// TIA Portal project "tank_level_control" (V17)

(* hardware
DEVICE "S7-1200 station_1"  S7-1200 Station
   slot 0: "Rack_0"  S7-1200 Rack  Rack  V1.0
   slot 1: "PLC_1"  CPU 1212C AC/DC/Rly  6ES7 212-1BE31-0XB0  V3.0
   slot 2: "DI 16x24VDC/DQ 16xRelay_1"  SM 1223 DI16/DQ16 x relay  6ES7 223-1PL32-0XB0  V2.0
DEVICE "HMI_1"  KTP600 Basic color PN
   slot 0: "HMI_1"  KTP600 Basic color PN  6AV6 647-0AD11-3AX0  12.0.0.0
   slot 1: "HMI_RT_1"  KTP600 Basic color PN  6AV6 647-0AD11-3AX0  12.0.0.0
   slot 5: "HMI_1.IE_CP_1"  PROFINET Interface  12.0.0.0
      slot 1: "PROFINET Interface_1"  PROFINET Interface
         slot 1: "Port_1"  Port
*)

// ===== PLC "PLC_1"  CPU 1212C AC/DC/Rly =====

VAR_GLOBAL   // PLC tag table "Default tag table"
   "OPEN" AT %M0.0 : Bool;
   "CLOSE" AT %M0.1 : Bool;
   "RUNNING" AT %Q0.2 : Bool;   // RUNNING LAMP INDICATOR
   "Tag_1" AT %M1.0 : Bool;
   "LEVEL" AT %MD100 : Real;
   "Tag_2" AT %MD102 : Real;
   "TANK_LEVEL" AT %MD90 : Real;
   "VALVE" AT %Q0.0 : Bool;
   "START" AT %M10.0 : Bool;
   "STOP" AT %M10.1 : Bool;
   "Tag_6" AT %M10.2 : Bool;
   "LL_LOW" AT %MD140 : Real;
   "LOW_LL_REACH" AT %M12.0 : Bool;
   "LL_HIGH" AT %MD144 : Real;
   "HIGH_LL_REACH" AT %M12.1 : Bool;
   "LL_LOW_BETTER" AT %MD156 : Real;
   "LL_HIGH_BETTER" AT %MD160 : Real;
END_VAR

// folder: System blocks/Program resources

DATA_BLOCK "T5"   // DB2
{ S7_Optimized_Access := 'TRUE' }
AUTHOR : Simatic
FAMILY : IEC
NAME : IEC_TMR
VERSION : 1.0
// stored: InstanceOfName IEC_TIMER
"IEC_TIMER"
BEGIN
END_DATA_BLOCK

DATA_BLOCK "T6"   // DB3
{ S7_Optimized_Access := 'TRUE' }
AUTHOR : Simatic
FAMILY : IEC
NAME : IEC_TMR
VERSION : 1.0
// stored: InstanceOfName IEC_TIMER
"IEC_TIMER"
BEGIN
END_DATA_BLOCK

// folder: (top level)

ORGANIZATION_BLOCK "Main"   // OB1, LAD, ProgramCycle
TITLE = "Main Program Sweep (Cycle)"
{ S7_Optimized_Access := 'TRUE' }
VERSION : 0.1
BEGIN

REGION Network 1: OPEN/CLOSE VALVE
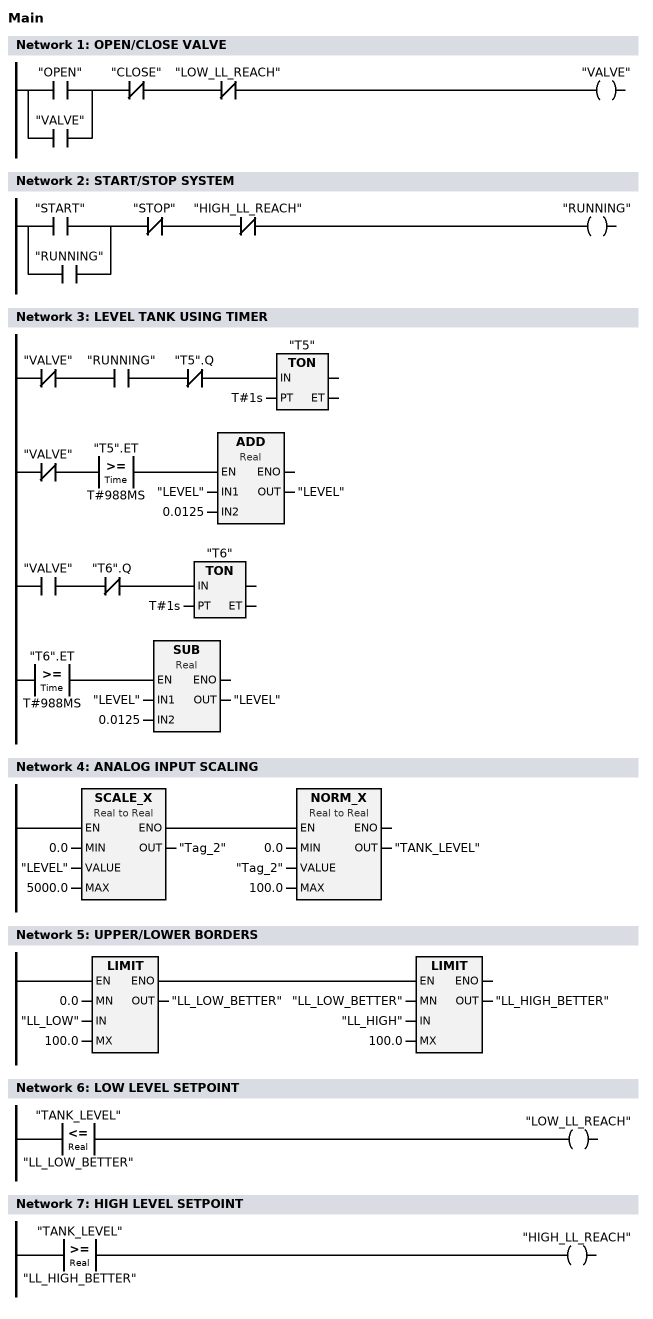
   RUNG wire#powerrail
      Contact( "OPEN" )
      wire#w1
      I_Contact( "CLOSE" )
      I_Contact( "LOW_LL_REACH" )
      Coil( "VALVE" )
   END_RUNG
   RUNG wire#powerrail
      Contact( "VALVE" )
   END_RUNG wire#w1
   // the same network as SCL:
   "VALVE" := ("OPEN" OR "VALVE") AND NOT "CLOSE" AND NOT "LOW_LL_REACH";
END_REGION

REGION Network 2: START/STOP SYSTEM
   RUNG wire#powerrail
      Contact( "START" )
      wire#w1
      I_Contact( "STOP" )
      I_Contact( "HIGH_LL_REACH" )
      Coil( "RUNNING" )
   END_RUNG
   RUNG wire#powerrail
      Contact( "RUNNING" )
   END_RUNG wire#w1
   // the same network as SCL:
   "RUNNING" := ("START" OR "RUNNING") AND NOT "STOP" AND NOT "HIGH_LL_REACH";
END_REGION

REGION Network 3: LEVEL TANK USING TIMER
   "T5".TON(IN := NOT "VALVE" AND "RUNNING" AND NOT "T5".Q, PT := T#1s);
   IF NOT "VALVE" AND ("T5".ET >= T#988MS) THEN "LEVEL" := "LEVEL" + 0.0125; END_IF;
   "T6".TON(IN := "VALVE" AND NOT "T6".Q, PT := T#1s);
   IF "T6".ET >= T#988MS THEN "LEVEL" := "LEVEL" - 0.0125; END_IF;
END_REGION

REGION Network 4: ANALOG INPUT SCALING
   RUNG wire#powerrail
      { S7_Templates := "[SrcType := Real, DestType := Real]"; S7_GenerateENO := "TRUE" } Scale(min := 0.0, value := "LEVEL", max := 5000.0, out => "Tag_2")
      { S7_Templates := "[SrcType := Real, DestType := Real]"; S7_GenerateENO := "TRUE" } Normalize(min := 0.0, value := "Tag_2", max := 100.0, out => "TANK_LEVEL")
   END_RUNG
   // the same network as SCL:
   // ENO of a box is taken as its EN; it also drops when the box reports an error
   "Tag_2" := SCALE_X(MIN := 0.0, VALUE := "LEVEL", MAX := 5000.0);
   "TANK_LEVEL" := NORM_X(MIN := 0.0, VALUE := "Tag_2", MAX := 100.0);
END_REGION

REGION Network 5: UPPER/LOWER BORDERS
   // ENO of a box is taken as its EN; it also drops when the box reports an error
   "LL_LOW_BETTER" := LIMIT(MN := 0.0, IN := "LL_LOW", MX := 100.0);
   "LL_HIGH_BETTER" := LIMIT(MN := "LL_LOW_BETTER", IN := "LL_HIGH", MX := 100.0);
END_REGION

REGION Network 6: LOW LEVEL SETPOINT
   RUNG wire#powerrail
      { S7_Templates := "SrcType := Real" } LE_Contact(in1 := "TANK_LEVEL", in2 := "LL_LOW_BETTER")
      Coil( "LOW_LL_REACH" )
   END_RUNG
   // the same network as SCL:
   "LOW_LL_REACH" := "TANK_LEVEL" <= "LL_LOW_BETTER";
END_REGION

REGION Network 7: HIGH LEVEL SETPOINT
   RUNG wire#powerrail
      { S7_Templates := "SrcType := Real" } GE_Contact(in1 := "TANK_LEVEL", in2 := "LL_HIGH_BETTER")
      Coil( "HIGH_LL_REACH" )
   END_RUNG
   // the same network as SCL:
   "HIGH_LL_REACH" := "TANK_LEVEL" >= "LL_HIGH_BETTER";
END_REGION
END_ORGANIZATION_BLOCK

(* ===== HMI "HMI_RT_1" =====
system functions are stored by id; their names below are inferred from use
connection "HMI_Connection_1": ETHERNET, SMART_S7_1200_OMS

HMI tags "Default tag table"
   "RUNNING" : Bool = PLC RUNNING AT %Q0.2, 1 s
   "START" : Bool = PLC START AT %M10.0, 1 s
   "STOP" : Bool = PLC STOP AT %M10.1, 1 s
   "OPEN" : Bool = PLC OPEN AT %M0.0, 1 s
   "CLOSE" : Bool = PLC CLOSE AT %M0.1, 1 s
   "LL_HIGH" : Real = PLC LL_HIGH AT %MD144, 1 s
   "LL_LOW" : Real = PLC LL_LOW AT %MD140, 1 s
   "TANK_LEVEL" : Real = PLC TANK_LEVEL AT %MD90, 1 s
   "LL_HIGH_BETTER" : Real = PLC LL_HIGH_BETTER AT %MD160, 1 s
   "VALVE" : Bool = PLC VALVE AT %Q0.0, 1 s

HMI tags "Second tag table"
   "TANK_LEVEL_BORDERS" : Real, internal

analog alarms
   1: 'Maximal value is 100%.', class Errors, trigger "LL_HIGH"
   2: 'Minimal value is 0%', class Errors, trigger "LL_LOW"

screen "Screen_1" 320x240
   TextField "Text field_1" at 172,6 size 137x18; Text 'TANK LEVEL CONTROL'
   Bar "Bar_1" at 213,92 size 81x120; MinimumValue 0; MaximumValue 100
      ProcessValue <- "TANK_LEVEL"
   Button "Button_1" at 15,6 size 50x23; TextOff 'START'
      on Press: SetBit("START")
      on Release: ResetBit("START")
   Button "Button_2" at 15,32 size 51x21; TextOff 'STOP'
      on Press: SetBit("STOP")
      on Release: ResetBit("STOP")
   Circle "Circle_1" at 100,11 size 20x20
      Appearance <- "RUNNING"
   IOField "I/O field_1" at 157,79 size 38x17; FormatPattern 9999
      ProcessValue <- "TANK_LEVEL"
   Button "Button_4" at 46,210 size 45x22; TextOff 'OPEN'
      on Press: SetBit("OPEN")
      on Release: ResetBit("OPEN")
   Button "Button_5" at 98,210 size 45x22; TextOff 'CLOSE'
      on Press: SetBit("CLOSE")
      on Release: ResetBit("CLOSE")
   TextField "Text field_3" at 121,62 size 76x13; Text 'LEVEL SENSOR'
   IOField "I/O field_2" at 95,119 size 49x17; FormatPattern 999.99
      ProcessValue <- "LL_HIGH"
   IOField "I/O field_3" at 95,139 size 49x17; FormatPattern 999.99
      ProcessValue <- "LL_LOW"
   TextField "Text field_2" at 17,120 size 74x13; Text 'UPPER LIMIT:'
   TextField "Text field_4" at 15,140 size 76x13; Text 'LOWER LIMIT:'
   Circle "Circle_2" at 166,175 size 20x20
      Appearance <- "VALVE"
   Button "Button_3" at 12,71 size 62x22; TextOff 'ALARMS'
      on Click: ActivateScreen("Screen_2", 0)

screen "Screen_2" 320x240
   AlarmView "Alarm view_1" at 0,0 size 319x239
   Button "Button_1" at 7,209 size 49x26; TextOff 'BACK'
      on Click: function_efd93a16()
   Button "Button_2" at 73,209 size 63x26; TextOff 'ARCHIVE'
      on Click: ActivateScreen("Screen_3", 0)

screen "Screen_3" 320x240
   AlarmView "Alarm view_1" at 0,0 size 319x239
   Button "Button_1" at 7,209 size 49x26; TextOff 'BACK'
      on Click: function_efd93a16()
*)